// Decides when FB_AstroClock may load the RTC blocks and whether the time can be trusted.
// Separate from FB_AstroClock so that it runs without ADS and can be unit tested.
//
// Feed it the Busy and Err outputs of NT_GetTime. The decision is taken at the moment Busy falls, because
// NT_GetTime raises Err in the same cycle: bSynchronize pulses for one cycle after a successful read only.
// A failed read must not load the RTCs, because the time structure it returns is stale (zero on the first call).
FUNCTION_BLOCK FB_AstroClockSync
VAR_INPUT
	bBusy			: BOOL;				// NT_GetTime.Busy
	bError			: BOOL;				// NT_GetTime.Err
END_VAR
VAR_OUTPUT
	bSynchronize	: BOOL;				// one cycle: load the RTCs from the time just read
	bValid			: BOOL;				// TRUE from the first successful read on; stays TRUE, the RTC keeps counting
	nErrors			: UINT;				// failed reads in a row (saturates at 65535), for diagnostics
END_VAR
VAR
	fbBusyDone		: F_TRIG;
	bEverSynchronized	: BOOL;
END_VAR

fbBusyDone(CLK := bBusy);
bSynchronize := FALSE;

IF fbBusyDone.Q THEN
	IF bError THEN
		IF nErrors < 65535 THEN
			nErrors := nErrors + 1;
		END_IF
	ELSE
		bSynchronize := TRUE;
		bEverSynchronized := TRUE;
		nErrors := 0;
	END_IF
END_IF

// After the first sync the RTC keeps counting on its own, so failed reads only make the last sync older (drift is
// far below a second over minutes). Only the time before the first sync is garbage, so that is all bValid excludes.
bValid := bEverSynchronized;

END_FUNCTION_BLOCK

(* stored: Version 1.1.0.1, ProductVersion 3.1.4024.15
   POU FB_AstroClockSync: Id {b7f0f43c-7ead-44a3-815d-4e88e648eb39}, SpecialFunc None *)
